PROGRAM PRG_CommandDispatcher
VAR
END_VAR

(* ---------------------------------------------------------
   程序骨架：HMI与Robot命令优先级、权限和事务仲裁。
   所属任务：Task_CffMain，调用顺序3。
   唯一Owner：PRG_CommandDispatcher。
   当前阶段：不产生Start/Stop/Initialize/Reset脉冲。
   后续实现：CommandId、Ack和单扫描内部Pulse。
   --------------------------------------------------------- *)

END_PROGRAM

(* stored: Version 1.1.0.1
   POU PRG_CommandDispatcher: Id {A2000000-0000-4000-8000-000000000007} *)
